TYPE VTD_Outputs_DUT :
STRUCT
	LP1_Retract:  BOOL;
	LP1_Extend:  BOOL;
	LP2_Retract:  Bool;
	LP2_Extend:  Bool;
	AE_Control_Word_1:  WORD;
	AE_Control_Word_2:  WORD;
END_STRUCT
END_TYPE

(* stored: Version 1.1.0.1
   DUT VTD_Outputs_DUT: Id {f7364db3-9ae9-4f02-af5e-df154e47a08a} *)
